// Mitsubishi GX Works2 project: RecipeMixerXDfix   PLC: FX3U/FX3UC

PROGRAM MAIN
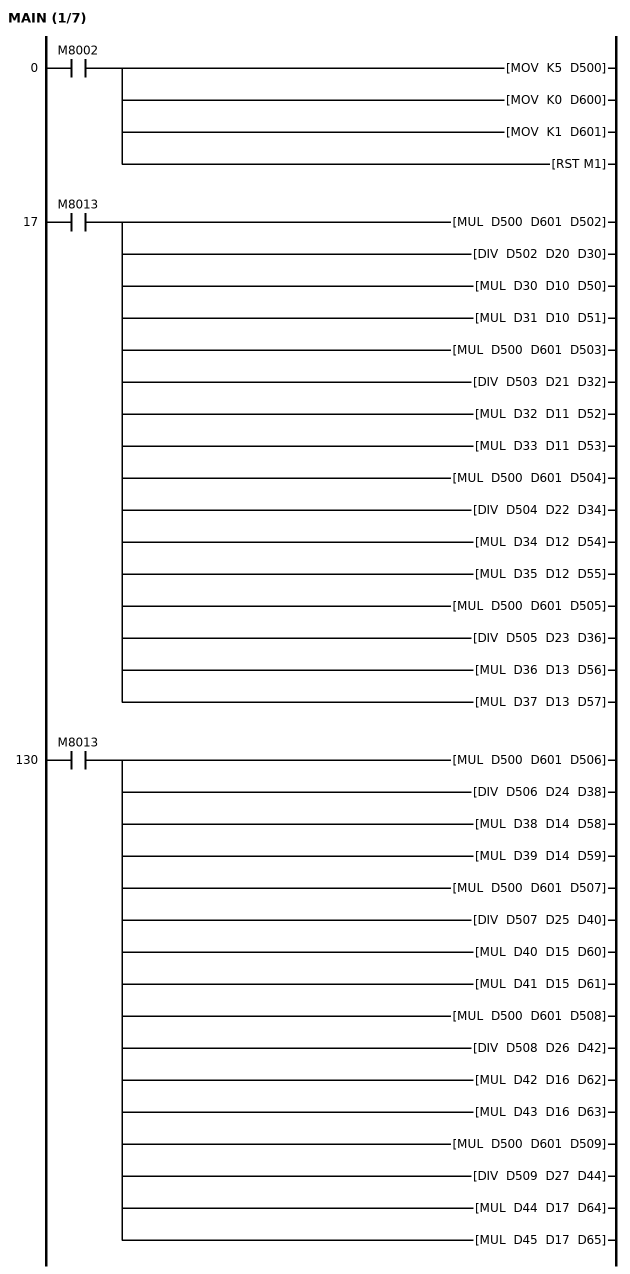
0     LD      M8002
      MOV     K5 D500
      MOV     K0 D600
      MOV     K1 D601
      RST     M1
17    LD      M8013
      MUL     D500 D601 D502
      DIV     D502 D20 D30
      MUL     D30 D10 D50
      MUL     D31 D10 D51
      MUL     D500 D601 D503
      DIV     D503 D21 D32
      MUL     D32 D11 D52
      MUL     D33 D11 D53
      MUL     D500 D601 D504
      DIV     D504 D22 D34
      MUL     D34 D12 D54
      MUL     D35 D12 D55
      MUL     D500 D601 D505
      DIV     D505 D23 D36
      MUL     D36 D13 D56
      MUL     D37 D13 D57
130   LD      M8013
      MUL     D500 D601 D506
      DIV     D506 D24 D38
      MUL     D38 D14 D58
      MUL     D39 D14 D59
      MUL     D500 D601 D507
      DIV     D507 D25 D40
      MUL     D40 D15 D60
      MUL     D41 D15 D61
      MUL     D500 D601 D508
      DIV     D508 D26 D42
      MUL     D42 D16 D62
      MUL     D43 D16 D63
      MUL     D500 D601 D509
      DIV     D509 D27 D44
      MUL     D44 D17 D64
      MUL     D45 D17 D65
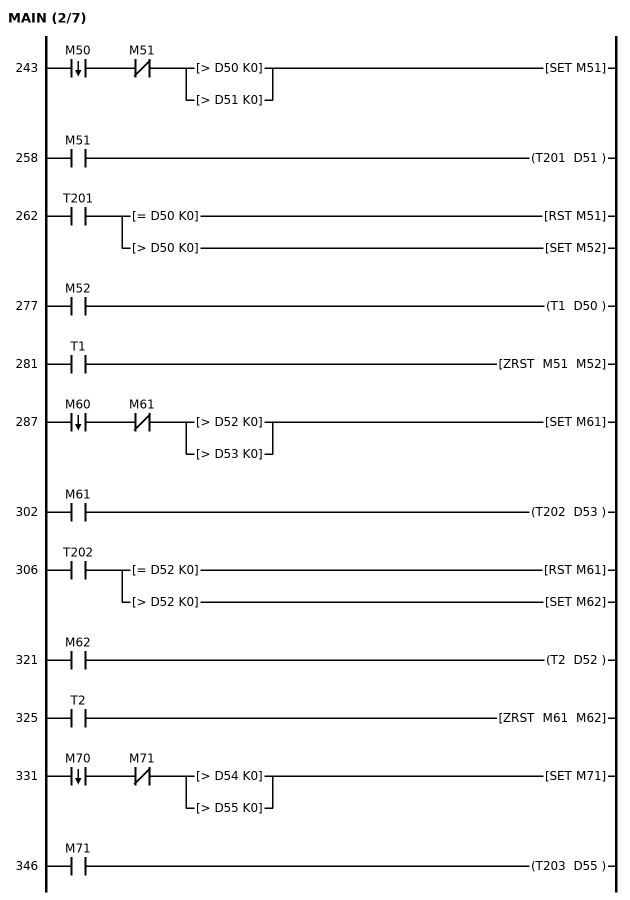
243   LDF     M50
      ANI     M51
      LD>     D50 K0
      OR>     D51 K0
      ANB
      SET     M51
258   LD      M51
      OUT     T201 D51
262   LD      T201
      MPS
      AND=    D50 K0
      RST     M51
      MPP
      AND>    D50 K0
      SET     M52
277   LD      M52
      OUT     T1 D50
281   LD      T1
      ZRST    M51 M52
287   LDF     M60
      ANI     M61
      LD>     D52 K0
      OR>     D53 K0
      ANB
      SET     M61
302   LD      M61
      OUT     T202 D53
306   LD      T202
      MPS
      AND=    D52 K0
      RST     M61
      MPP
      AND>    D52 K0
      SET     M62
321   LD      M62
      OUT     T2 D52
325   LD      T2
      ZRST    M61 M62
331   LDF     M70
      ANI     M71
      LD>     D54 K0
      OR>     D55 K0
      ANB
      SET     M71
346   LD      M71
      OUT     T203 D55
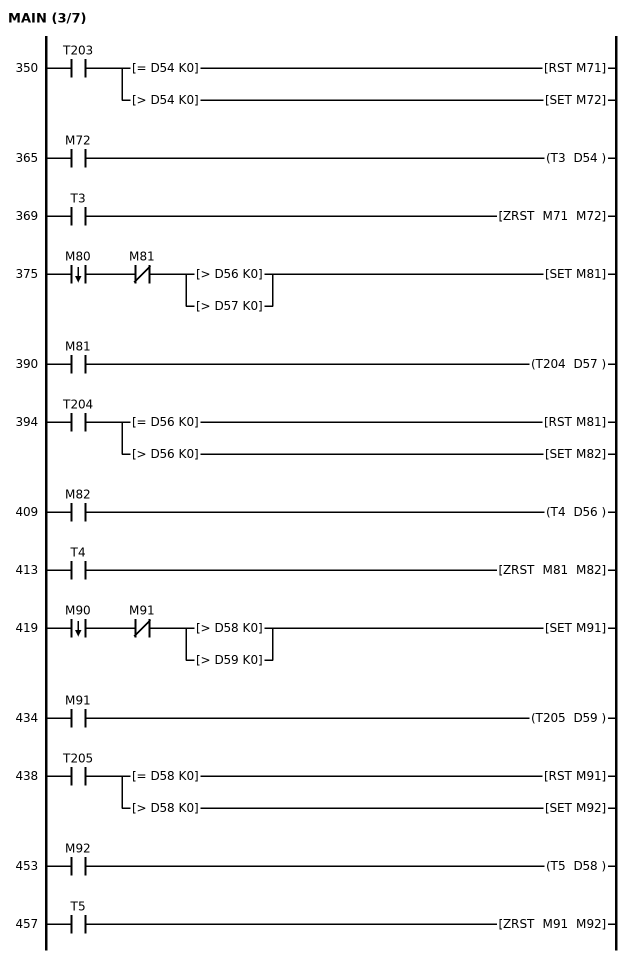
350   LD      T203
      MPS
      AND=    D54 K0
      RST     M71
      MPP
      AND>    D54 K0
      SET     M72
365   LD      M72
      OUT     T3 D54
369   LD      T3
      ZRST    M71 M72
375   LDF     M80
      ANI     M81
      LD>     D56 K0
      OR>     D57 K0
      ANB
      SET     M81
390   LD      M81
      OUT     T204 D57
394   LD      T204
      MPS
      AND=    D56 K0
      RST     M81
      MPP
      AND>    D56 K0
      SET     M82
409   LD      M82
      OUT     T4 D56
413   LD      T4
      ZRST    M81 M82
419   LDF     M90
      ANI     M91
      LD>     D58 K0
      OR>     D59 K0
      ANB
      SET     M91
434   LD      M91
      OUT     T205 D59
438   LD      T205
      MPS
      AND=    D58 K0
      RST     M91
      MPP
      AND>    D58 K0
      SET     M92
453   LD      M92
      OUT     T5 D58
457   LD      T5
      ZRST    M91 M92
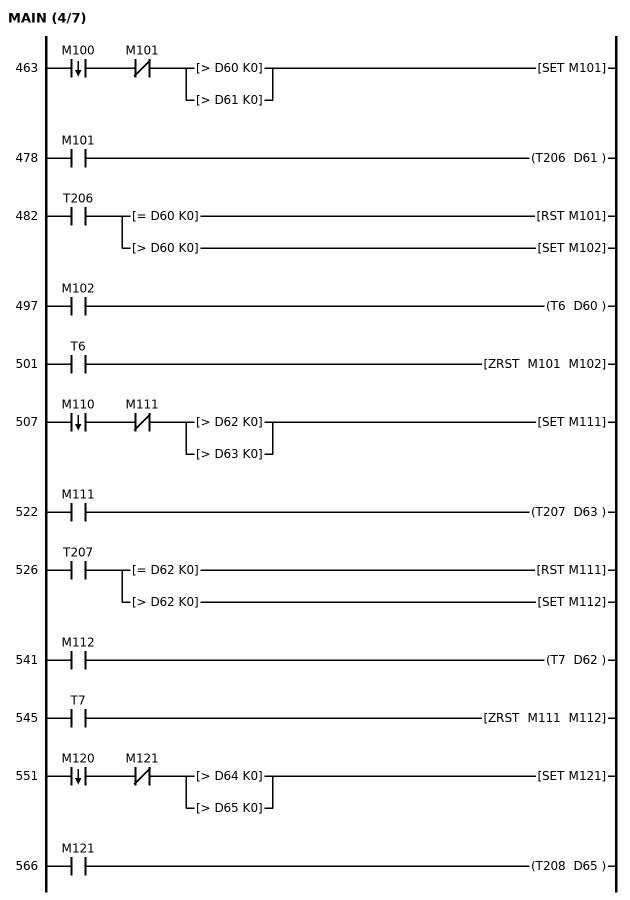
463   LDF     M100
      ANI     M101
      LD>     D60 K0
      OR>     D61 K0
      ANB
      SET     M101
478   LD      M101
      OUT     T206 D61
482   LD      T206
      MPS
      AND=    D60 K0
      RST     M101
      MPP
      AND>    D60 K0
      SET     M102
497   LD      M102
      OUT     T6 D60
501   LD      T6
      ZRST    M101 M102
507   LDF     M110
      ANI     M111
      LD>     D62 K0
      OR>     D63 K0
      ANB
      SET     M111
522   LD      M111
      OUT     T207 D63
526   LD      T207
      MPS
      AND=    D62 K0
      RST     M111
      MPP
      AND>    D62 K0
      SET     M112
541   LD      M112
      OUT     T7 D62
545   LD      T7
      ZRST    M111 M112
551   LDF     M120
      ANI     M121
      LD>     D64 K0
      OR>     D65 K0
      ANB
      SET     M121
566   LD      M121
      OUT     T208 D65
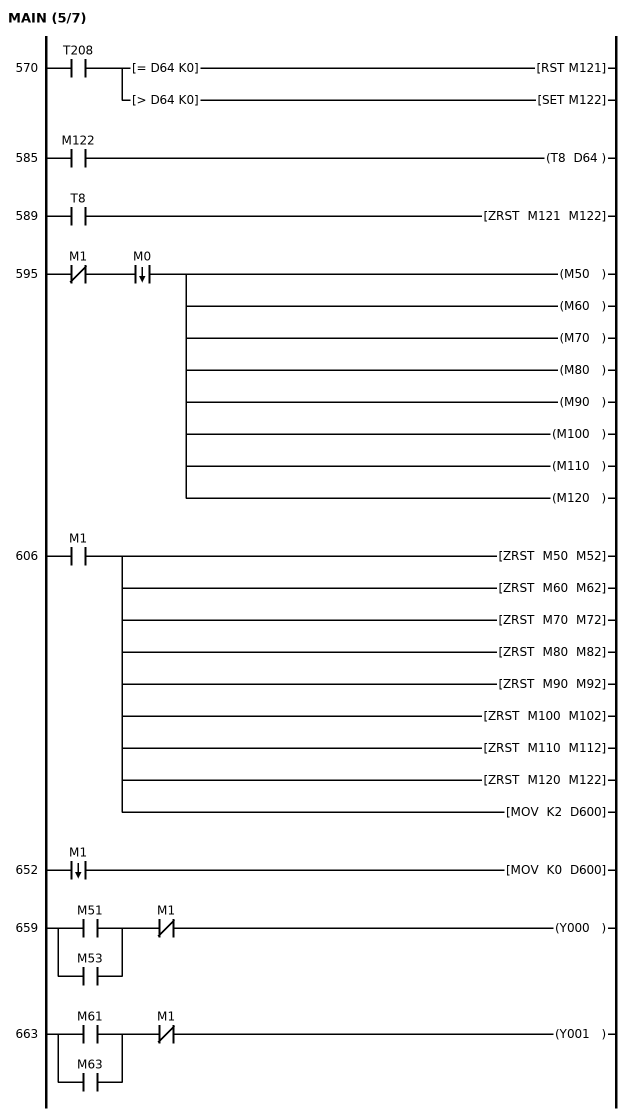
570   LD      T208
      MPS
      AND=    D64 K0
      RST     M121
      MPP
      AND>    D64 K0
      SET     M122
585   LD      M122
      OUT     T8 D64
589   LD      T8
      ZRST    M121 M122
595   LDI     M1
      ANDF    M0
      OUT     M50
      OUT     M60
      OUT     M70
      OUT     M80
      OUT     M90
      OUT     M100
      OUT     M110
      OUT     M120
606   LD      M1
      ZRST    M50 M52
      ZRST    M60 M62
      ZRST    M70 M72
      ZRST    M80 M82
      ZRST    M90 M92
      ZRST    M100 M102
      ZRST    M110 M112
      ZRST    M120 M122
      MOV     K2 D600
652   LDF     M1
      MOV     K0 D600
659   LD      M51
      OR      M53
      ANI     M1
      OUT     Y000
663   LD      M61
      OR      M63
      ANI     M1
      OUT     Y001
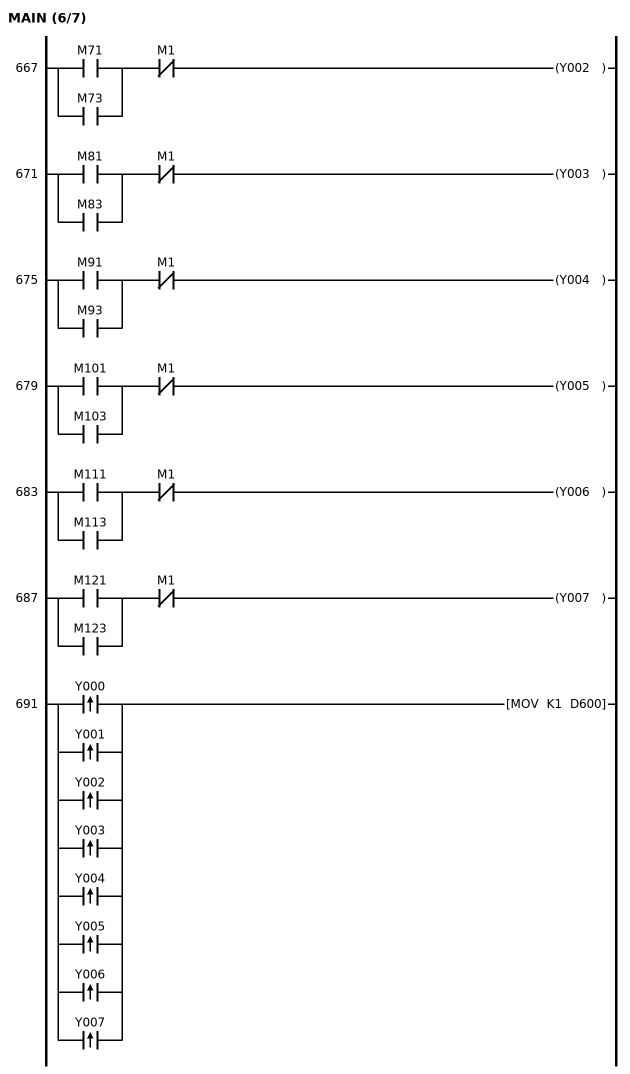
667   LD      M71
      OR      M73
      ANI     M1
      OUT     Y002
671   LD      M81
      OR      M83
      ANI     M1
      OUT     Y003
675   LD      M91
      OR      M93
      ANI     M1
      OUT     Y004
679   LD      M101
      OR      M103
      ANI     M1
      OUT     Y005
683   LD      M111
      OR      M113
      ANI     M1
      OUT     Y006
687   LD      M121
      OR      M123
      ANI     M1
      OUT     Y007
691   LDP     Y000
      ORP     Y001
      ORP     Y002
      ORP     Y003
      ORP     Y004
      ORP     Y005
      ORP     Y006
      ORP     Y007
      MOV     K1 D600
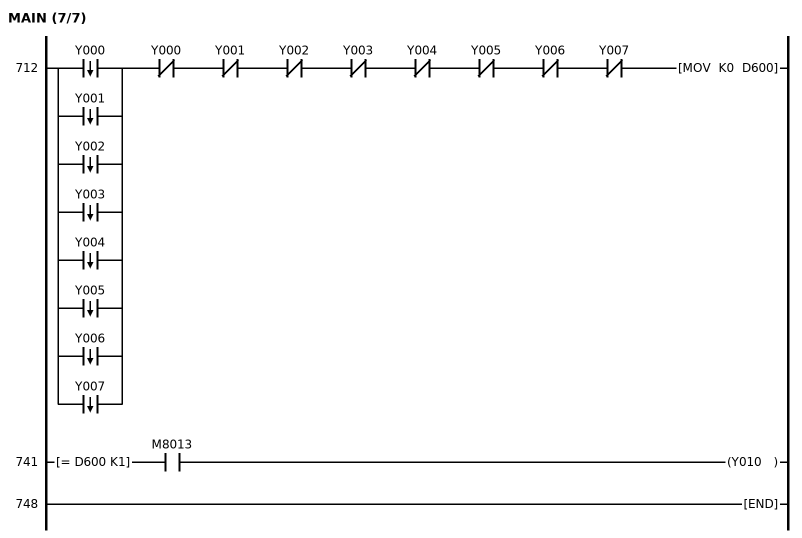
712   LDF     Y000
      ORF     Y001
      ORF     Y002
      ORF     Y003
      ORF     Y004
      ORF     Y005
      ORF     Y006
      ORF     Y007
      ANI     Y000
      ANI     Y001
      ANI     Y002
      ANI     Y003
      ANI     Y004
      ANI     Y005
      ANI     Y006
      ANI     Y007
      MOV     K0 D600
741   LD=     D600 K1
      AND     M8013
      OUT     Y010
748   END
END_PROGRAM
